// TIA Portal V20 export
FUNCTION "PlantAutoControl" : Void   // FC100, LAD
TITLE = Plant Automatic Control
// Per-equipment automatic-control layer for the shredding/material-recovery plant (REQ-001..022). Paradigm: combinational chained-permissive interlock/mapping (C-113 'no' - no phase memory in this block; the plant sequencer and equipment FBs hold the state). One network per machine, in material-train order, each mapping field feedback in, computing the auto start/shutdown permissives from PlantControl.Status and neighbour UPSEnable/ShutdownComplete, driving the physical output, and calling the equipment FB. Composed from the chained-permissive-enable pattern. Net 17 (feed conveyor) is freeform fwd/rev per C-116/C-117 (reversal pause enforced inside MotorFwdRevSystem). Author: lad-coder (gen-block-new). Rev 1, 2026-07-20.
BEGIN

REGION Network 1: Incline Feed Conveyor Automatic Control
   // Incline feed VSD (MotorVSDInst2). Running-fwd confirmation taken from the rotation sensor (inferred VSD-running mapping - review). Holds during shutdown until the link conveyor and the third-party JOB9001 plant have both completed shutdown (REQ-003/014); starts once the air-separator VSD is enabled (REQ-004).
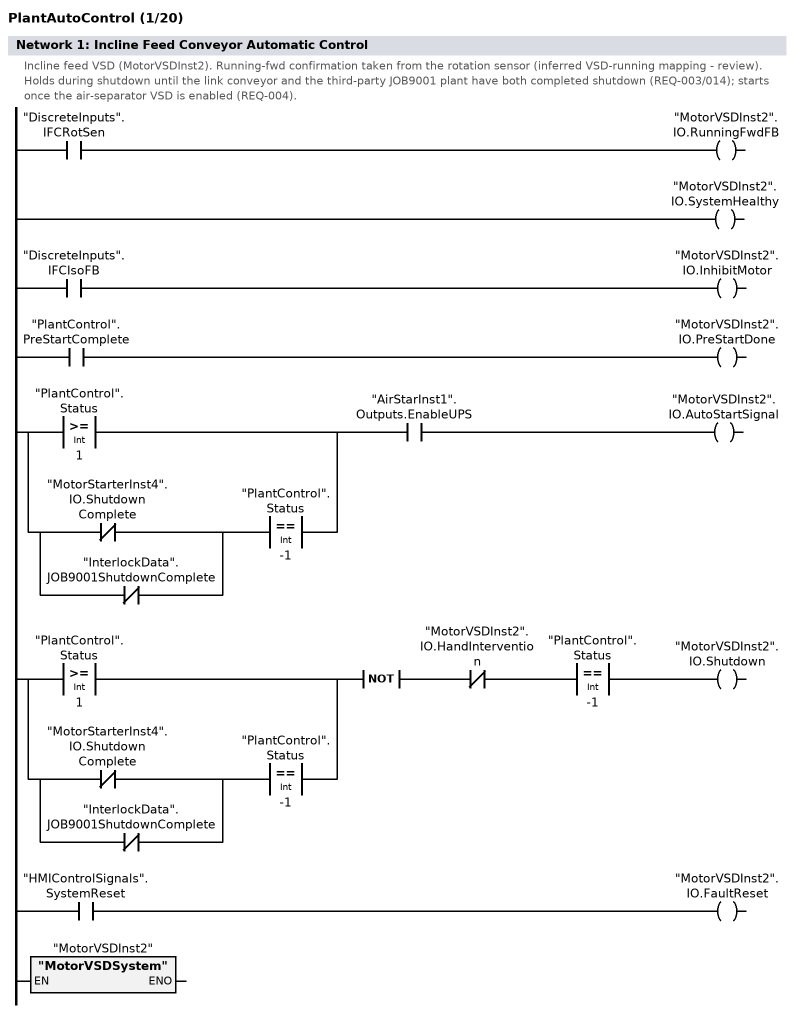
   "MotorVSDInst2".IO.RunningFwdFB := "DiscreteInputs".IFCRotSen;
   "MotorVSDInst2".IO.SystemHealthy := TRUE;
   "MotorVSDInst2".IO.InhibitMotor := "DiscreteInputs".IFCIsoFB;
   "MotorVSDInst2".IO.PreStartDone := "PlantControl".PreStartComplete;
   "MotorVSDInst2".IO.AutoStartSignal := (("PlantControl".Status >= 1) OR ((NOT "MotorStarterInst4".IO.ShutdownComplete OR NOT "InterlockData".JOB9001ShutdownComplete) AND ("PlantControl".Status = (-1)))) AND "AirStarInst1".Outputs.EnableUPS;
   "MotorVSDInst2".IO.Shutdown := NOT (("PlantControl".Status >= 1) OR ((NOT "MotorStarterInst4".IO.ShutdownComplete OR NOT "InterlockData".JOB9001ShutdownComplete) AND ("PlantControl".Status = (-1)))) AND NOT "MotorVSDInst2".IO.HandIntervention AND ("PlantControl".Status = (-1));
   "MotorVSDInst2".IO.FaultReset := "HMIControlSignals".SystemReset;
   "MotorVSDInst2"();   // "MotorVSDSystem"
END_REGION

REGION Network 2: Link Conveyor Automatic Control
   // Link conveyor (MotorStarterInst4), the designated first machine. Gated by the third-party JOB9001 interlock; holds through shutdown until JOB9001 signals its own shutdown complete (REQ-014). On first auto-start it requests the plant pre-start warning once (one-shot via PlantControl.PositiveEdgeArray[4]), cleared when the pre-start output energises (REQ-015).
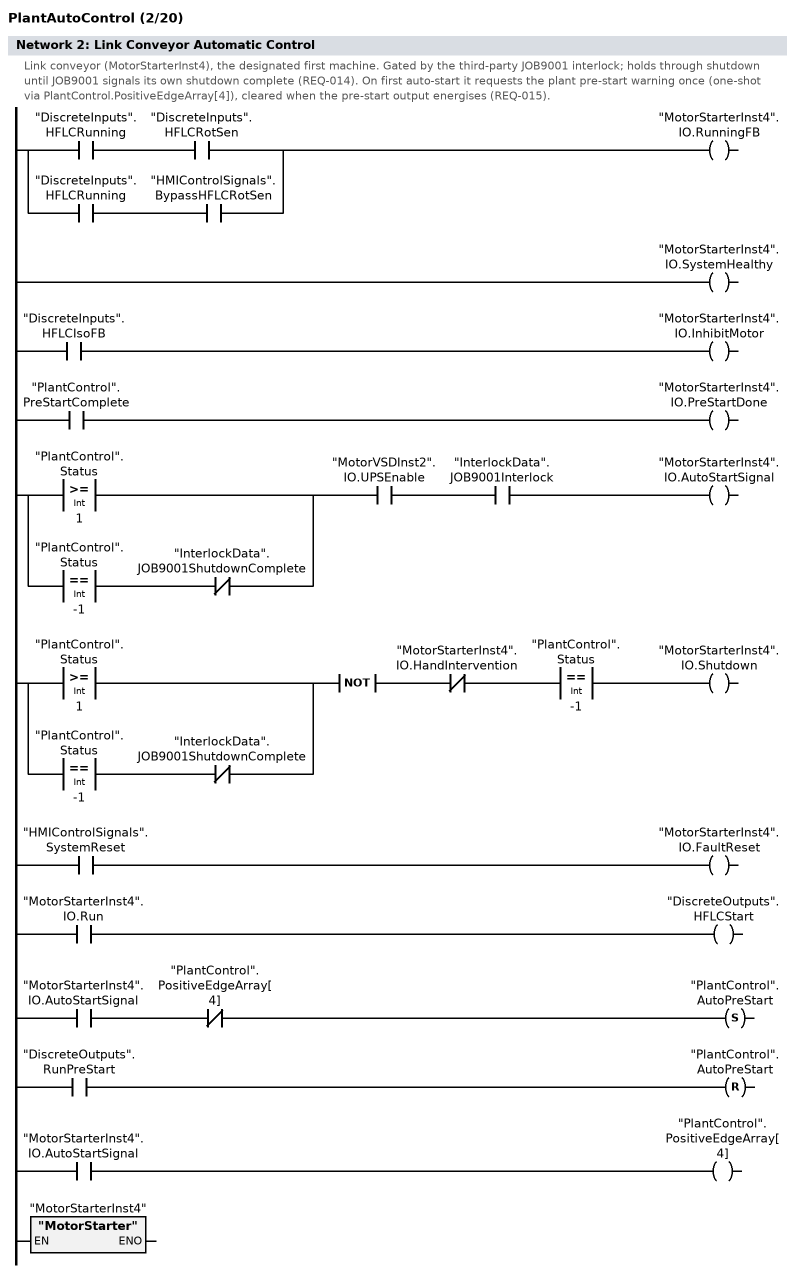
   "MotorStarterInst4".IO.RunningFB := ("DiscreteInputs".HFLCRunning AND "DiscreteInputs".HFLCRotSen) OR ("DiscreteInputs".HFLCRunning AND "HMIControlSignals".BypassHFLCRotSen);
   "MotorStarterInst4".IO.SystemHealthy := TRUE;
   "MotorStarterInst4".IO.InhibitMotor := "DiscreteInputs".HFLCIsoFB;
   "MotorStarterInst4".IO.PreStartDone := "PlantControl".PreStartComplete;
   "MotorStarterInst4".IO.AutoStartSignal := (("PlantControl".Status >= 1) OR (("PlantControl".Status = (-1)) AND NOT "InterlockData".JOB9001ShutdownComplete)) AND "MotorVSDInst2".IO.UPSEnable AND "InterlockData".JOB9001Interlock;
   "MotorStarterInst4".IO.Shutdown := NOT (("PlantControl".Status >= 1) OR (("PlantControl".Status = (-1)) AND NOT "InterlockData".JOB9001ShutdownComplete)) AND NOT "MotorStarterInst4".IO.HandIntervention AND ("PlantControl".Status = (-1));
   "MotorStarterInst4".IO.FaultReset := "HMIControlSignals".SystemReset;
   "DiscreteOutputs".HFLCStart := "MotorStarterInst4".IO.Run;
   IF "MotorStarterInst4".IO.AutoStartSignal AND NOT "PlantControl".PositiveEdgeArray[4] THEN
       "PlantControl".AutoPreStart := TRUE;
   END_IF;
   IF "DiscreteOutputs".RunPreStart THEN "PlantControl".AutoPreStart := FALSE; END_IF;
   "PlantControl".PositiveEdgeArray[4] := "MotorStarterInst4".IO.AutoStartSignal;
   "MotorStarterInst4"();   // "MotorStarter"
END_REGION

REGION Network 3: Dust Filter Unit 1 Automatic Control
   // Dust filter unit 1 (FilterUnitInst2). Remote-operational, running(=ready) and fault feedbacks brought in; fault reset echoed to the physical unit (REQ-019). Fan up-to-speed delay set from the plant fan-start time (REQ-020); see block header re C-308. Starts once the sorter conveyor VSD is enabled; holds during shutdown until fans-shutdown-ready (REQ-003/013).
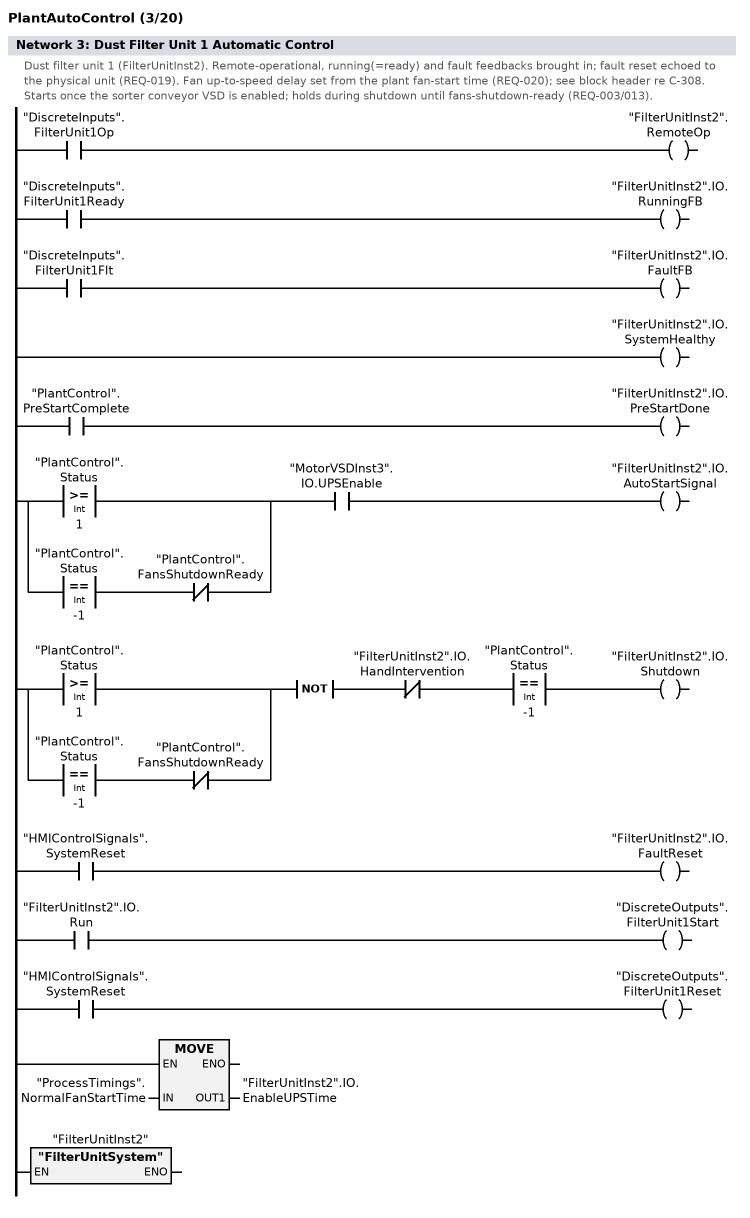
   "FilterUnitInst2".RemoteOp := "DiscreteInputs".FilterUnit1Op;
   "FilterUnitInst2".IO.RunningFB := "DiscreteInputs".FilterUnit1Ready;
   "FilterUnitInst2".IO.FaultFB := "DiscreteInputs".FilterUnit1Flt;
   "FilterUnitInst2".IO.SystemHealthy := TRUE;
   "FilterUnitInst2".IO.PreStartDone := "PlantControl".PreStartComplete;
   "FilterUnitInst2".IO.AutoStartSignal := (("PlantControl".Status >= 1) OR (("PlantControl".Status = (-1)) AND NOT "PlantControl".FansShutdownReady)) AND "MotorVSDInst3".IO.UPSEnable;
   "FilterUnitInst2".IO.Shutdown := NOT (("PlantControl".Status >= 1) OR (("PlantControl".Status = (-1)) AND NOT "PlantControl".FansShutdownReady)) AND NOT "FilterUnitInst2".IO.HandIntervention AND ("PlantControl".Status = (-1));
   "FilterUnitInst2".IO.FaultReset := "HMIControlSignals".SystemReset;
   "DiscreteOutputs".FilterUnit1Start := "FilterUnitInst2".IO.Run;
   "DiscreteOutputs".FilterUnit1Reset := "HMIControlSignals".SystemReset;
   "FilterUnitInst2".IO.EnableUPSTime := "ProcessTimings".NormalFanStartTime;
   "FilterUnitInst2"();   // "FilterUnitSystem"
END_REGION

REGION Network 4: Dust Filter Unit 2 Automatic Control
   // Dust filter unit 2 (FilterUnitInst3), identical shape to unit 1 (REQ-019/020). Starts once the sorter conveyor VSD is enabled; holds until fans-shutdown-ready.
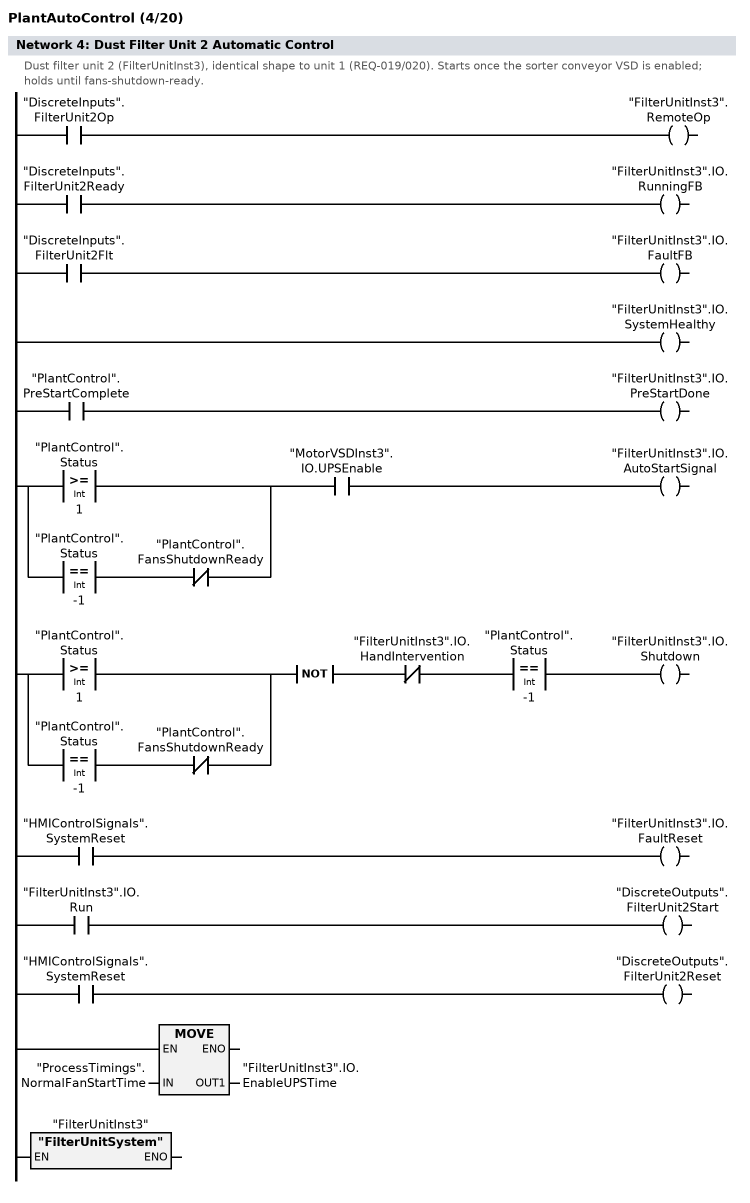
   "FilterUnitInst3".RemoteOp := "DiscreteInputs".FilterUnit2Op;
   "FilterUnitInst3".IO.RunningFB := "DiscreteInputs".FilterUnit2Ready;
   "FilterUnitInst3".IO.FaultFB := "DiscreteInputs".FilterUnit2Flt;
   "FilterUnitInst3".IO.SystemHealthy := TRUE;
   "FilterUnitInst3".IO.PreStartDone := "PlantControl".PreStartComplete;
   "FilterUnitInst3".IO.AutoStartSignal := (("PlantControl".Status >= 1) OR (("PlantControl".Status = (-1)) AND NOT "PlantControl".FansShutdownReady)) AND "MotorVSDInst3".IO.UPSEnable;
   "FilterUnitInst3".IO.Shutdown := NOT (("PlantControl".Status >= 1) OR (("PlantControl".Status = (-1)) AND NOT "PlantControl".FansShutdownReady)) AND NOT "FilterUnitInst3".IO.HandIntervention AND ("PlantControl".Status = (-1));
   "FilterUnitInst3".IO.FaultReset := "HMIControlSignals".SystemReset;
   "DiscreteOutputs".FilterUnit2Start := "FilterUnitInst3".IO.Run;
   "DiscreteOutputs".FilterUnit2Reset := "HMIControlSignals".SystemReset;
   "FilterUnitInst3".IO.EnableUPSTime := "ProcessTimings".NormalFanStartTime;
   "FilterUnitInst3"();   // "FilterUnitSystem"
END_REGION

REGION Network 5: Air-Separator VSD Automatic Control
   // Air-separator VSD (AirStarInst1), a bus-coupled drive with no discrete start output. Running confirmed over comms (MachineRunning). Alternative start permissive: discharge-conveyor VSD plus both dust filters enabled, OR discharge-conveyor VSD plus the third-party link-out signal (REQ-021). Holds during shutdown until the incline feed conveyor has shut down (REQ-003).
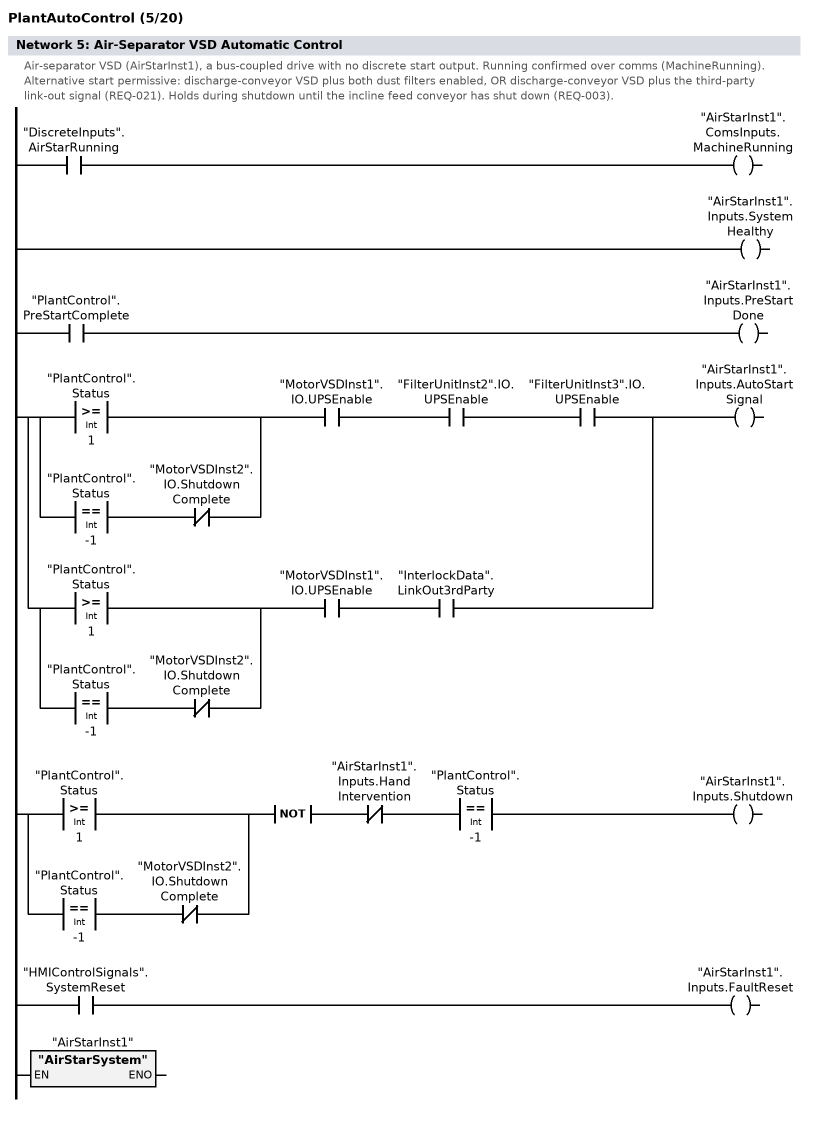
   "AirStarInst1".ComsInputs.MachineRunning := "DiscreteInputs".AirStarRunning;
   "AirStarInst1".Inputs.SystemHealthy := TRUE;
   "AirStarInst1".Inputs.PreStartDone := "PlantControl".PreStartComplete;
   "AirStarInst1".Inputs.AutoStartSignal := ((("PlantControl".Status >= 1) OR (("PlantControl".Status = (-1)) AND NOT "MotorVSDInst2".IO.ShutdownComplete)) AND "MotorVSDInst1".IO.UPSEnable AND "FilterUnitInst2".IO.UPSEnable AND "FilterUnitInst3".IO.UPSEnable) OR ((("PlantControl".Status >= 1) OR (("PlantControl".Status = (-1)) AND NOT "MotorVSDInst2".IO.ShutdownComplete)) AND "MotorVSDInst1".IO.UPSEnable AND "InterlockData".LinkOut3rdParty);
   "AirStarInst1".Inputs.Shutdown := NOT (("PlantControl".Status >= 1) OR (("PlantControl".Status = (-1)) AND NOT "MotorVSDInst2".IO.ShutdownComplete)) AND NOT "AirStarInst1".Inputs.HandIntervention AND ("PlantControl".Status = (-1));
   "AirStarInst1".Inputs.FaultReset := "HMIControlSignals".SystemReset;
   "AirStarInst1"();   // "AirStarSystem"
END_REGION

REGION Network 6: Discharge Conveyor VSD Automatic Control
   // Discharge conveyor VSD (MotorVSDInst1). Treats its rotation sensor as running-forward confirmation (REQ-012; bypass handling deferred - review). Starts once the overband magnet and ECS are enabled; holds during shutdown until the air-separator VSD has shut down (REQ-003/004).
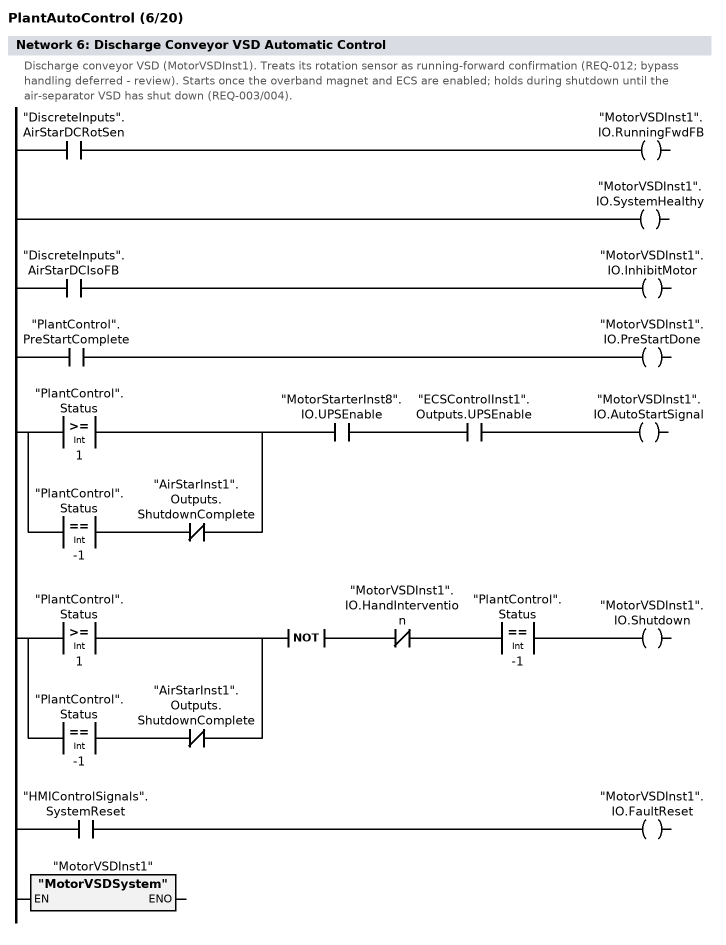
   "MotorVSDInst1".IO.RunningFwdFB := "DiscreteInputs".AirStarDCRotSen;
   "MotorVSDInst1".IO.SystemHealthy := TRUE;
   "MotorVSDInst1".IO.InhibitMotor := "DiscreteInputs".AirStarDCIsoFB;
   "MotorVSDInst1".IO.PreStartDone := "PlantControl".PreStartComplete;
   "MotorVSDInst1".IO.AutoStartSignal := (("PlantControl".Status >= 1) OR (("PlantControl".Status = (-1)) AND NOT "AirStarInst1".Outputs.ShutdownComplete)) AND "MotorStarterInst8".IO.UPSEnable AND "ECSControlInst1".Outputs.UPSEnable;
   "MotorVSDInst1".IO.Shutdown := NOT (("PlantControl".Status >= 1) OR (("PlantControl".Status = (-1)) AND NOT "AirStarInst1".Outputs.ShutdownComplete)) AND NOT "MotorVSDInst1".IO.HandIntervention AND ("PlantControl".Status = (-1));
   "MotorVSDInst1".IO.FaultReset := "HMIControlSignals".SystemReset;
   "MotorVSDInst1"();   // "MotorVSDSystem"
END_REGION

REGION Network 7: Metal Collection Conveyor Automatic Control
   // Metal collection conveyor (MotorStarterInst3). Gated by the magnet-circuit enable (REQ-013); starts on that plant flag rather than an upstream UPSEnable. Holds during shutdown until the overband magnet has shut down (REQ-003).
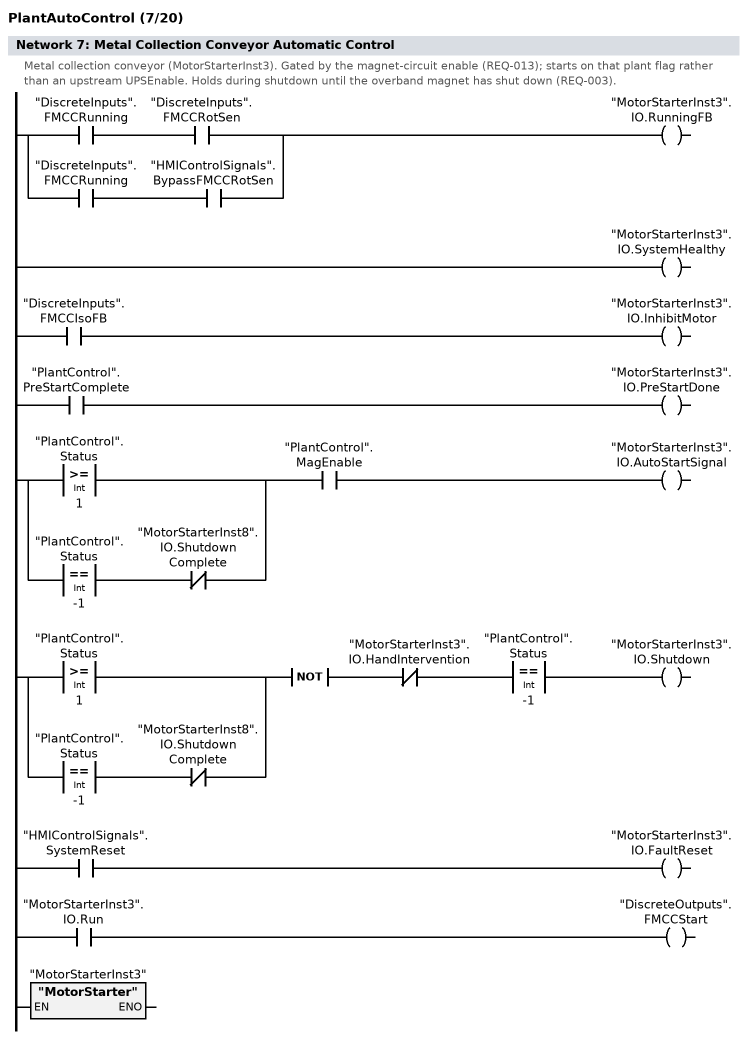
   "MotorStarterInst3".IO.RunningFB := ("DiscreteInputs".FMCCRunning AND "DiscreteInputs".FMCCRotSen) OR ("DiscreteInputs".FMCCRunning AND "HMIControlSignals".BypassFMCCRotSen);
   "MotorStarterInst3".IO.SystemHealthy := TRUE;
   "MotorStarterInst3".IO.InhibitMotor := "DiscreteInputs".FMCCIsoFB;
   "MotorStarterInst3".IO.PreStartDone := "PlantControl".PreStartComplete;
   "MotorStarterInst3".IO.AutoStartSignal := (("PlantControl".Status >= 1) OR (("PlantControl".Status = (-1)) AND NOT "MotorStarterInst8".IO.ShutdownComplete)) AND "PlantControl".MagEnable;
   "MotorStarterInst3".IO.Shutdown := NOT (("PlantControl".Status >= 1) OR (("PlantControl".Status = (-1)) AND NOT "MotorStarterInst8".IO.ShutdownComplete)) AND NOT "MotorStarterInst3".IO.HandIntervention AND ("PlantControl".Status = (-1));
   "MotorStarterInst3".IO.FaultReset := "HMIControlSignals".SystemReset;
   "DiscreteOutputs".FMCCStart := "MotorStarterInst3".IO.Run;
   "MotorStarterInst3"();   // "MotorStarter"
END_REGION

REGION Network 8: Overband Magnet Automatic Control
   // Overband magnet (MotorStarterInst8), confirmed on run feedback only (no rotation sensor). Starts once the metal collection conveyor is enabled; holds during shutdown until the discharge conveyor VSD has shut down (REQ-003/004).
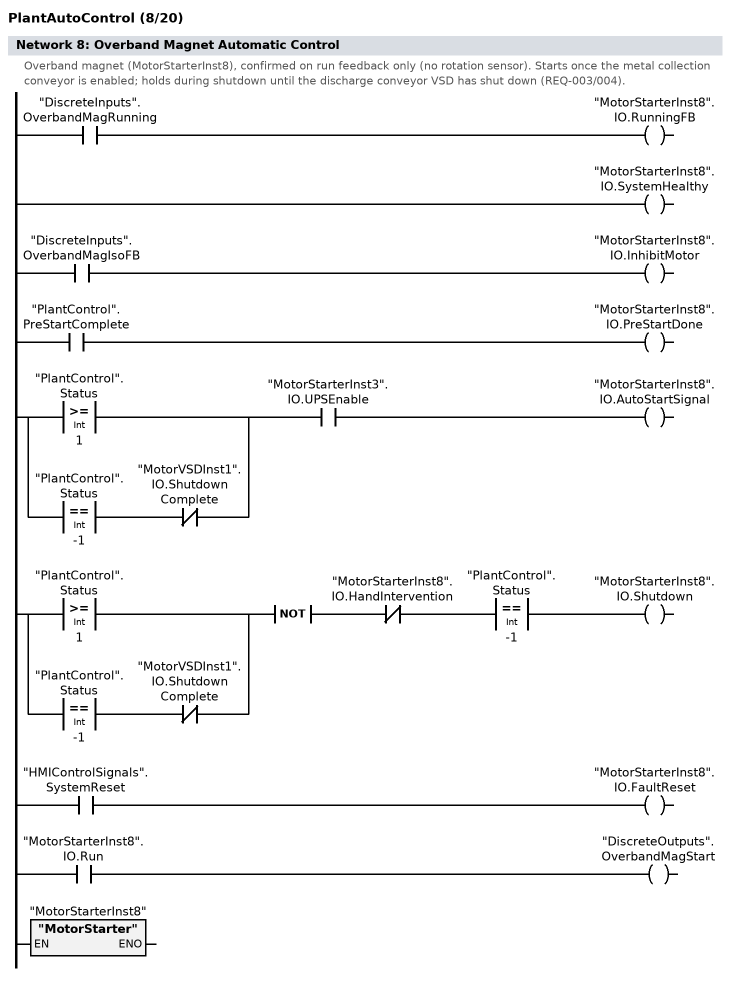
   "MotorStarterInst8".IO.RunningFB := "DiscreteInputs".OverbandMagRunning;
   "MotorStarterInst8".IO.SystemHealthy := TRUE;
   "MotorStarterInst8".IO.InhibitMotor := "DiscreteInputs".OverbandMagIsoFB;
   "MotorStarterInst8".IO.PreStartDone := "PlantControl".PreStartComplete;
   "MotorStarterInst8".IO.AutoStartSignal := (("PlantControl".Status >= 1) OR (("PlantControl".Status = (-1)) AND NOT "MotorVSDInst1".IO.ShutdownComplete)) AND "MotorStarterInst3".IO.UPSEnable;
   "MotorStarterInst8".IO.Shutdown := NOT (("PlantControl".Status >= 1) OR (("PlantControl".Status = (-1)) AND NOT "MotorVSDInst1".IO.ShutdownComplete)) AND NOT "MotorStarterInst8".IO.HandIntervention AND ("PlantControl".Status = (-1));
   "MotorStarterInst8".IO.FaultReset := "HMIControlSignals".SystemReset;
   "DiscreteOutputs".OverbandMagStart := "MotorStarterInst8".IO.Run;
   "MotorStarterInst8"();   // "MotorStarter"
END_REGION

REGION Network 9: Equipment Control System Automatic Control
   // Equipment control system (ECSControlInst1). Fault, mode (auto/hand/setting), ready, running, feeder/charge and rotor status brought in; auto-start and reset outputs driven (REQ-018). Starts once the sorter conveyor VSD is enabled; holds during shutdown until the discharge conveyor VSD has shut down (REQ-003).
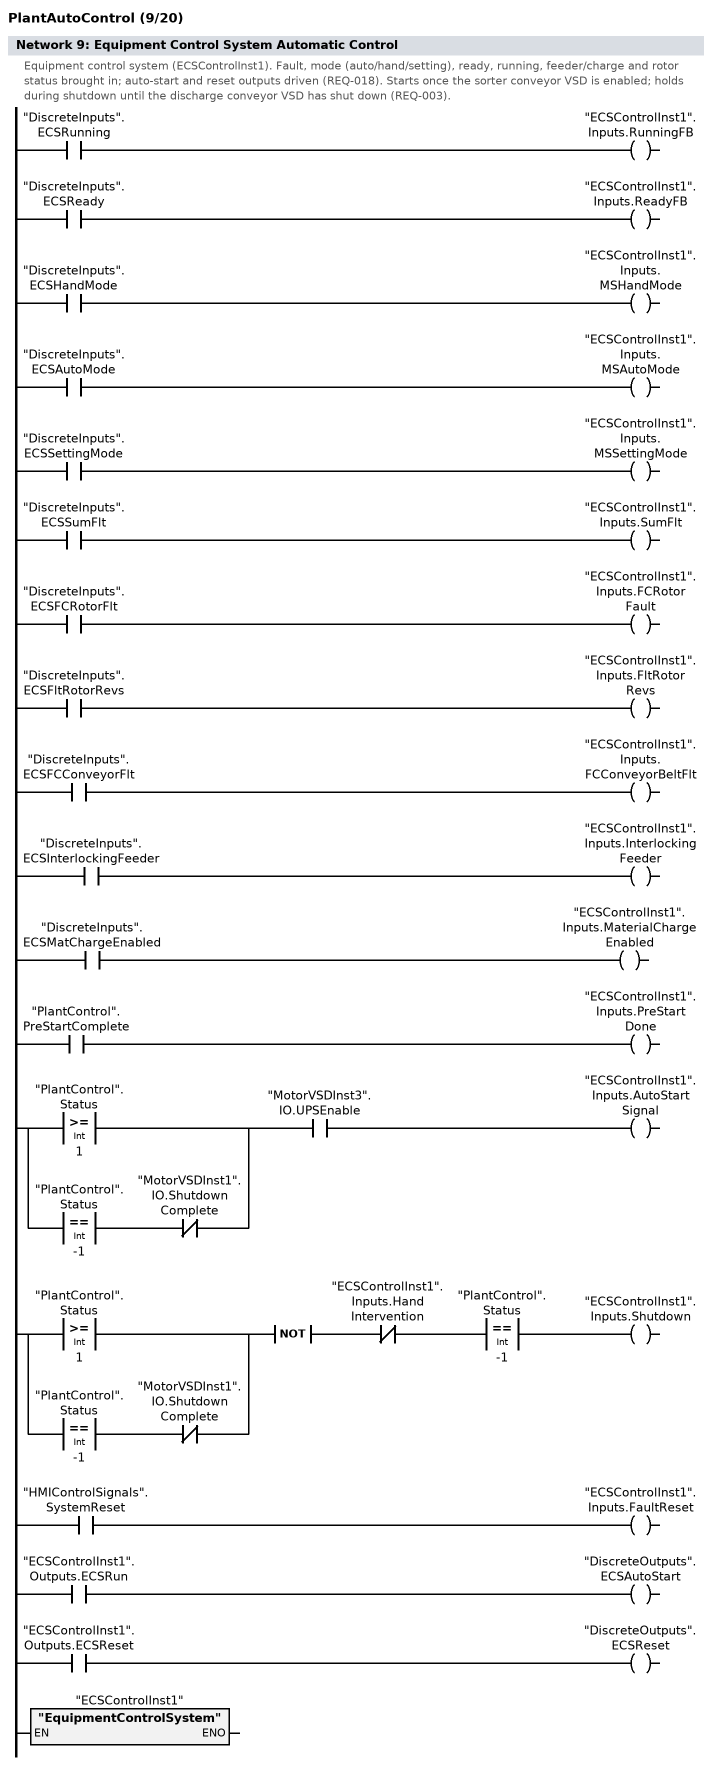
   "ECSControlInst1".Inputs.RunningFB := "DiscreteInputs".ECSRunning;
   "ECSControlInst1".Inputs.ReadyFB := "DiscreteInputs".ECSReady;
   "ECSControlInst1".Inputs.MSHandMode := "DiscreteInputs".ECSHandMode;
   "ECSControlInst1".Inputs.MSAutoMode := "DiscreteInputs".ECSAutoMode;
   "ECSControlInst1".Inputs.MSSettingMode := "DiscreteInputs".ECSSettingMode;
   "ECSControlInst1".Inputs.SumFlt := "DiscreteInputs".ECSSumFlt;
   "ECSControlInst1".Inputs.FCRotorFault := "DiscreteInputs".ECSFCRotorFlt;
   "ECSControlInst1".Inputs.FltRotorRevs := "DiscreteInputs".ECSFltRotorRevs;
   "ECSControlInst1".Inputs.FCConveyorBeltFlt := "DiscreteInputs".ECSFCConveyorFlt;
   "ECSControlInst1".Inputs.InterlockingFeeder := "DiscreteInputs".ECSInterlockingFeeder;
   "ECSControlInst1".Inputs.MaterialChargeEnabled := "DiscreteInputs".ECSMatChargeEnabled;
   "ECSControlInst1".Inputs.PreStartDone := "PlantControl".PreStartComplete;
   "ECSControlInst1".Inputs.AutoStartSignal := (("PlantControl".Status >= 1) OR (("PlantControl".Status = (-1)) AND NOT "MotorVSDInst1".IO.ShutdownComplete)) AND "MotorVSDInst3".IO.UPSEnable;
   "ECSControlInst1".Inputs.Shutdown := NOT (("PlantControl".Status >= 1) OR (("PlantControl".Status = (-1)) AND NOT "MotorVSDInst1".IO.ShutdownComplete)) AND NOT "ECSControlInst1".Inputs.HandIntervention AND ("PlantControl".Status = (-1));
   "ECSControlInst1".Inputs.FaultReset := "HMIControlSignals".SystemReset;
   "DiscreteOutputs".ECSAutoStart := "ECSControlInst1".Outputs.ECSRun;
   "DiscreteOutputs".ECSReset := "ECSControlInst1".Outputs.ECSReset;
   "ECSControlInst1"();   // "EquipmentControlSystem"
END_REGION

REGION Network 10: Sorter Conveyor VSD Automatic Control
   // Sorter feed conveyor VSD (MotorVSDInst3). Running-fwd from rotation sensor (inferred - review). Only permitted to start while the optical sorter is ready and not faulted, and the ejected and residual conveyors are enabled (REQ-017/004). Holds during shutdown until the ECS has shut down (REQ-003).
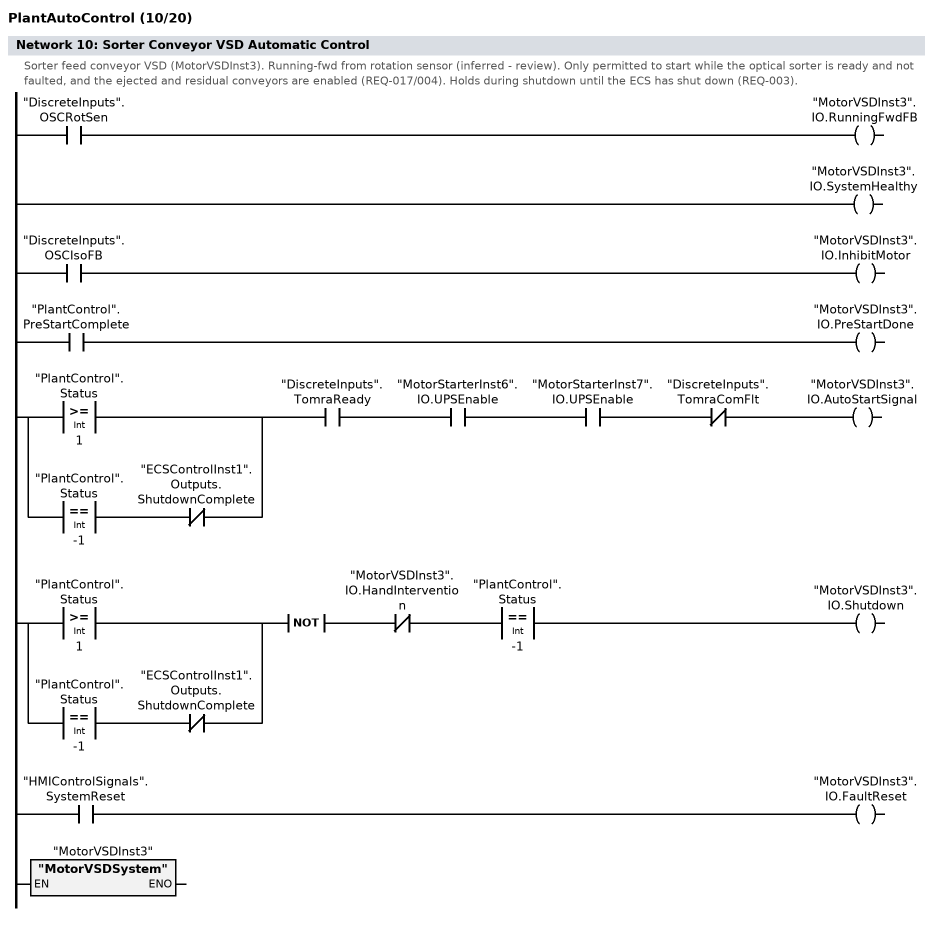
   "MotorVSDInst3".IO.RunningFwdFB := "DiscreteInputs".OSCRotSen;
   "MotorVSDInst3".IO.SystemHealthy := TRUE;
   "MotorVSDInst3".IO.InhibitMotor := "DiscreteInputs".OSCIsoFB;
   "MotorVSDInst3".IO.PreStartDone := "PlantControl".PreStartComplete;
   "MotorVSDInst3".IO.AutoStartSignal := (("PlantControl".Status >= 1) OR (("PlantControl".Status = (-1)) AND NOT "ECSControlInst1".Outputs.ShutdownComplete)) AND "DiscreteInputs".TomraReady AND "MotorStarterInst6".IO.UPSEnable AND "MotorStarterInst7".IO.UPSEnable AND NOT "DiscreteInputs".TomraComFlt;
   "MotorVSDInst3".IO.Shutdown := NOT (("PlantControl".Status >= 1) OR (("PlantControl".Status = (-1)) AND NOT "ECSControlInst1".Outputs.ShutdownComplete)) AND NOT "MotorVSDInst3".IO.HandIntervention AND ("PlantControl".Status = (-1));
   "MotorVSDInst3".IO.FaultReset := "HMIControlSignals".SystemReset;
   "MotorVSDInst3"();   // "MotorVSDSystem"
END_REGION

REGION Network 11: Optical Sorter Automatic Control
   // Optical sorter (TomraControlInst1). Hardwired ready/running/comms-fault brought in and the run command driven to the sorter (REQ-017). Comms data words (a separate block owns them) deliberately not wired here. Starts once the ejected and residual conveyors are enabled; holds during shutdown until the sorter conveyor VSD has shut down (REQ-003).
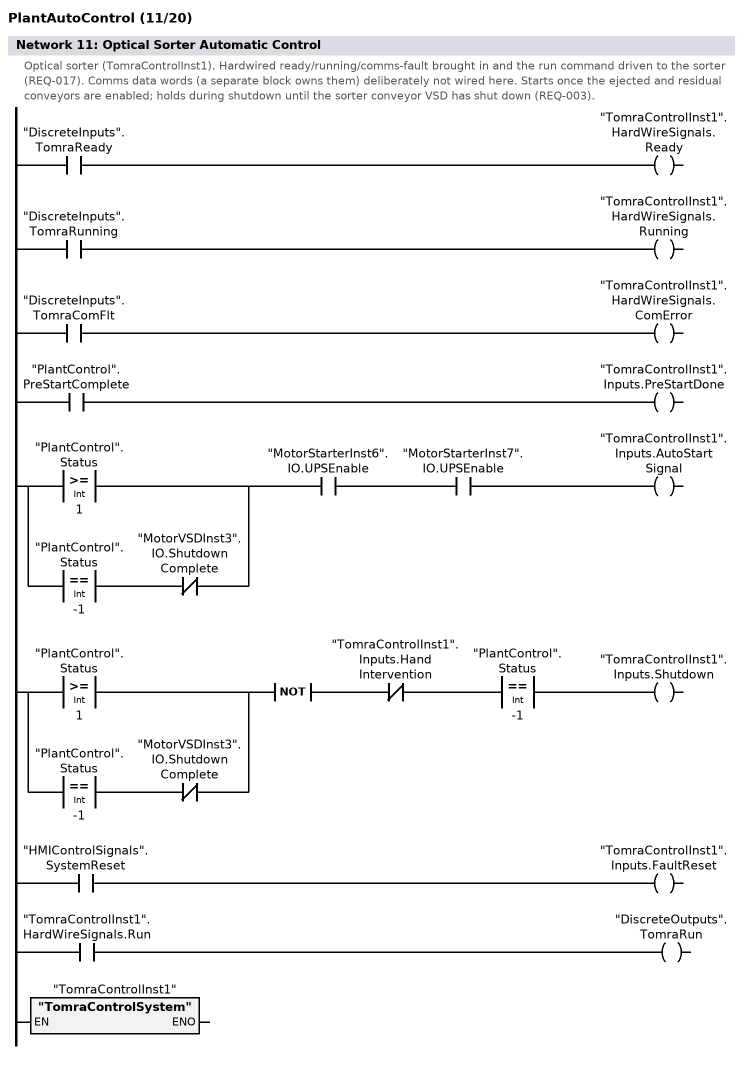
   "TomraControlInst1".HardWireSignals.Ready := "DiscreteInputs".TomraReady;
   "TomraControlInst1".HardWireSignals.Running := "DiscreteInputs".TomraRunning;
   "TomraControlInst1".HardWireSignals.ComError := "DiscreteInputs".TomraComFlt;
   "TomraControlInst1".Inputs.PreStartDone := "PlantControl".PreStartComplete;
   "TomraControlInst1".Inputs.AutoStartSignal := (("PlantControl".Status >= 1) OR (("PlantControl".Status = (-1)) AND NOT "MotorVSDInst3".IO.ShutdownComplete)) AND "MotorStarterInst6".IO.UPSEnable AND "MotorStarterInst7".IO.UPSEnable;
   "TomraControlInst1".Inputs.Shutdown := NOT (("PlantControl".Status >= 1) OR (("PlantControl".Status = (-1)) AND NOT "MotorVSDInst3".IO.ShutdownComplete)) AND NOT "TomraControlInst1".Inputs.HandIntervention AND ("PlantControl".Status = (-1));
   "TomraControlInst1".Inputs.FaultReset := "HMIControlSignals".SystemReset;
   "DiscreteOutputs".TomraRun := "TomraControlInst1".HardWireSignals.Run;
   "TomraControlInst1"();   // "TomraControlSystem"
END_REGION

REGION Network 12: Drum Separator Automatic Control
   // Drum separator (MotorStarterInst5), confirmed on run feedback only. Gated by the drum-separator enable (REQ-013); holds during shutdown until drum-shutdown-ready (REQ-003).
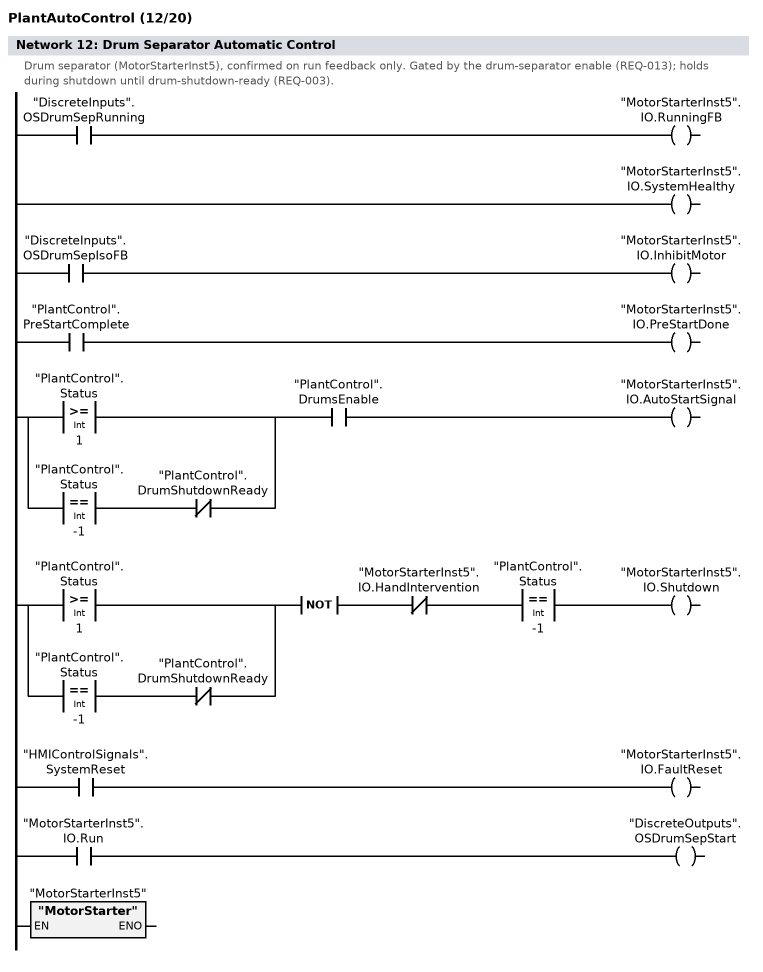
   "MotorStarterInst5".IO.RunningFB := "DiscreteInputs".OSDrumSepRunning;
   "MotorStarterInst5".IO.SystemHealthy := TRUE;
   "MotorStarterInst5".IO.InhibitMotor := "DiscreteInputs".OSDrumSepIsoFB;
   "MotorStarterInst5".IO.PreStartDone := "PlantControl".PreStartComplete;
   "MotorStarterInst5".IO.AutoStartSignal := (("PlantControl".Status >= 1) OR (("PlantControl".Status = (-1)) AND NOT "PlantControl".DrumShutdownReady)) AND "PlantControl".DrumsEnable;
   "MotorStarterInst5".IO.Shutdown := NOT (("PlantControl".Status >= 1) OR (("PlantControl".Status = (-1)) AND NOT "PlantControl".DrumShutdownReady)) AND NOT "MotorStarterInst5".IO.HandIntervention AND ("PlantControl".Status = (-1));
   "MotorStarterInst5".IO.FaultReset := "HMIControlSignals".SystemReset;
   "DiscreteOutputs".OSDrumSepStart := "MotorStarterInst5".IO.Run;
   "MotorStarterInst5"();   // "MotorStarter"
END_REGION

REGION Network 13: Ejected Material Conveyor Automatic Control
   // Ejected material conveyor (MotorStarterInst6). Gated by the general enable (REQ-013); holds during shutdown until the optical sorter has shut down (REQ-003).
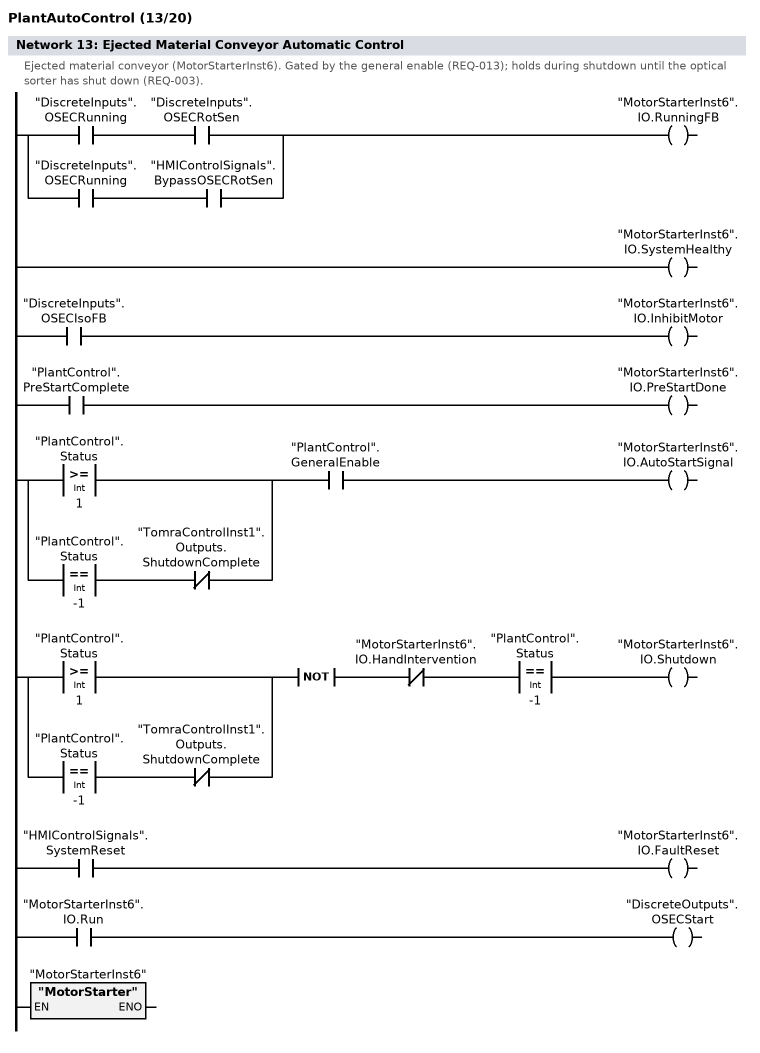
   "MotorStarterInst6".IO.RunningFB := ("DiscreteInputs".OSECRunning AND "DiscreteInputs".OSECRotSen) OR ("DiscreteInputs".OSECRunning AND "HMIControlSignals".BypassOSECRotSen);
   "MotorStarterInst6".IO.SystemHealthy := TRUE;
   "MotorStarterInst6".IO.InhibitMotor := "DiscreteInputs".OSECIsoFB;
   "MotorStarterInst6".IO.PreStartDone := "PlantControl".PreStartComplete;
   "MotorStarterInst6".IO.AutoStartSignal := (("PlantControl".Status >= 1) OR (("PlantControl".Status = (-1)) AND NOT "TomraControlInst1".Outputs.ShutdownComplete)) AND "PlantControl".GeneralEnable;
   "MotorStarterInst6".IO.Shutdown := NOT (("PlantControl".Status >= 1) OR (("PlantControl".Status = (-1)) AND NOT "TomraControlInst1".Outputs.ShutdownComplete)) AND NOT "MotorStarterInst6".IO.HandIntervention AND ("PlantControl".Status = (-1));
   "MotorStarterInst6".IO.FaultReset := "HMIControlSignals".SystemReset;
   "DiscreteOutputs".OSECStart := "MotorStarterInst6".IO.Run;
   "MotorStarterInst6"();   // "MotorStarter"
END_REGION

REGION Network 14: Residual Material Conveyor Automatic Control
   // Residual material conveyor (MotorStarterInst7). Starts once disc spreaders 1 and 2 are enabled; holds during shutdown until the optical sorter has shut down (REQ-003/004).
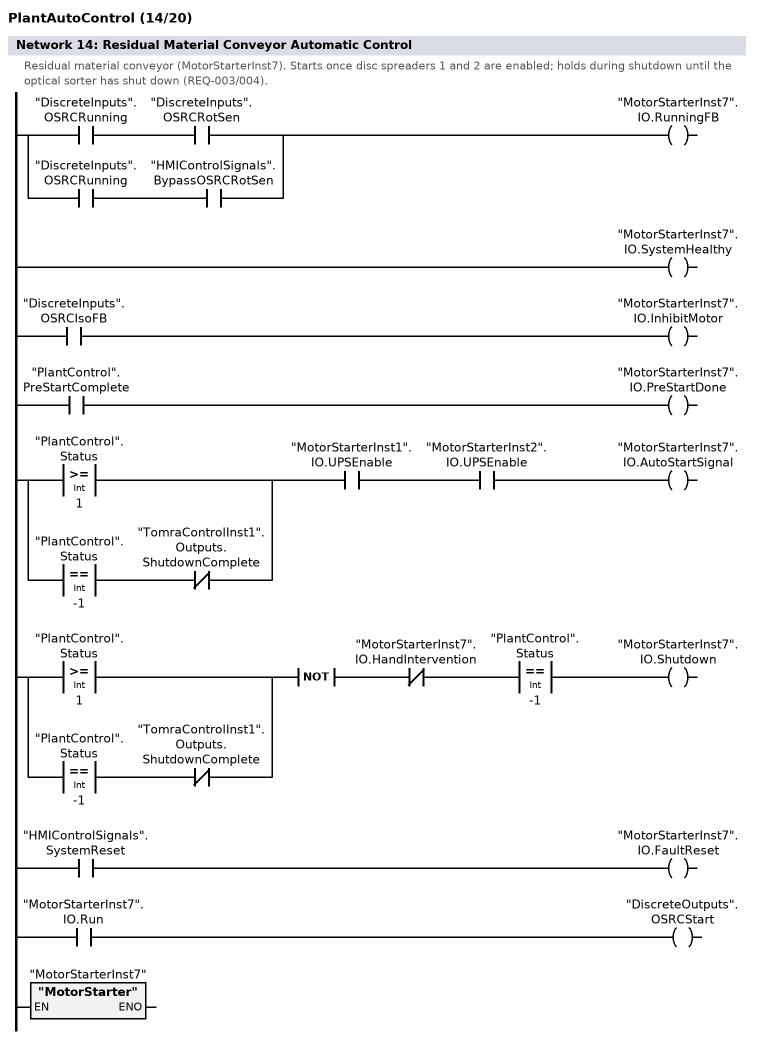
   "MotorStarterInst7".IO.RunningFB := ("DiscreteInputs".OSRCRunning AND "DiscreteInputs".OSRCRotSen) OR ("DiscreteInputs".OSRCRunning AND "HMIControlSignals".BypassOSRCRotSen);
   "MotorStarterInst7".IO.SystemHealthy := TRUE;
   "MotorStarterInst7".IO.InhibitMotor := "DiscreteInputs".OSRCIsoFB;
   "MotorStarterInst7".IO.PreStartDone := "PlantControl".PreStartComplete;
   "MotorStarterInst7".IO.AutoStartSignal := (("PlantControl".Status >= 1) OR (("PlantControl".Status = (-1)) AND NOT "TomraControlInst1".Outputs.ShutdownComplete)) AND "MotorStarterInst1".IO.UPSEnable AND "MotorStarterInst2".IO.UPSEnable;
   "MotorStarterInst7".IO.Shutdown := NOT (("PlantControl".Status >= 1) OR (("PlantControl".Status = (-1)) AND NOT "TomraControlInst1".Outputs.ShutdownComplete)) AND NOT "MotorStarterInst7".IO.HandIntervention AND ("PlantControl".Status = (-1));
   "MotorStarterInst7".IO.FaultReset := "HMIControlSignals".SystemReset;
   "DiscreteOutputs".OSRCStart := "MotorStarterInst7".IO.Run;
   "MotorStarterInst7"();   // "MotorStarter"
END_REGION

REGION Network 15: Disc Spreader Unit 1 Automatic Control
   // Disc spreader unit 1 (MotorStarterInst1), confirmed on run feedback only. Starts once the feed conveyor is enabled; holds during shutdown until the residual material conveyor has shut down (REQ-003/004).
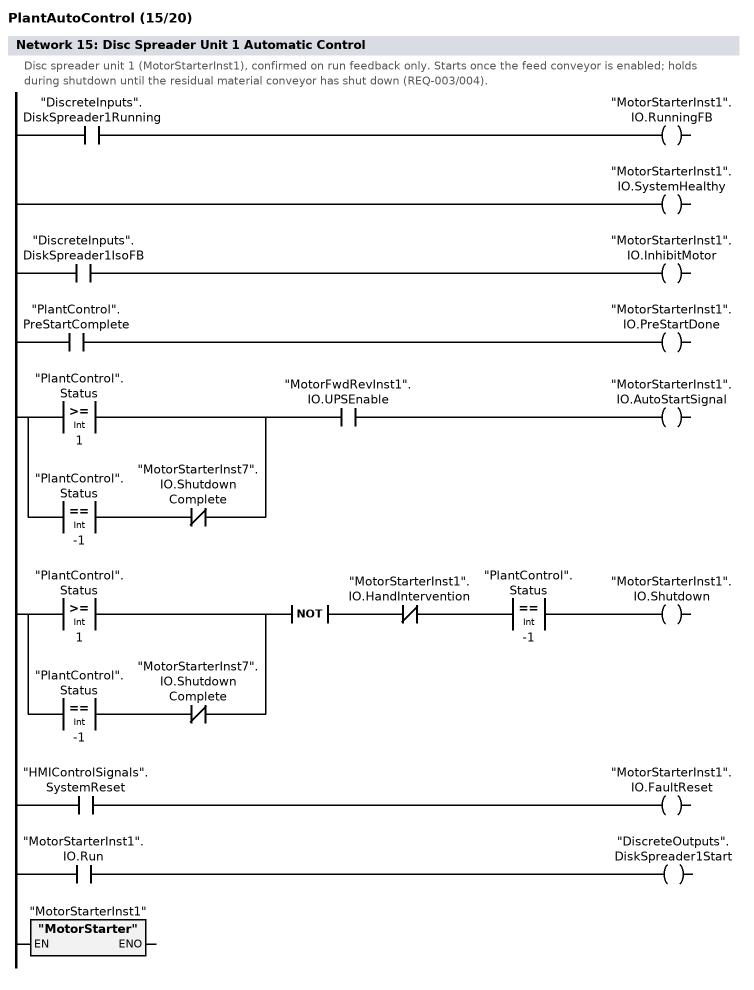
   "MotorStarterInst1".IO.RunningFB := "DiscreteInputs".DiskSpreader1Running;
   "MotorStarterInst1".IO.SystemHealthy := TRUE;
   "MotorStarterInst1".IO.InhibitMotor := "DiscreteInputs".DiskSpreader1IsoFB;
   "MotorStarterInst1".IO.PreStartDone := "PlantControl".PreStartComplete;
   "MotorStarterInst1".IO.AutoStartSignal := (("PlantControl".Status >= 1) OR (("PlantControl".Status = (-1)) AND NOT "MotorStarterInst7".IO.ShutdownComplete)) AND "MotorFwdRevInst1".IO.UPSEnable;
   "MotorStarterInst1".IO.Shutdown := NOT (("PlantControl".Status >= 1) OR (("PlantControl".Status = (-1)) AND NOT "MotorStarterInst7".IO.ShutdownComplete)) AND NOT "MotorStarterInst1".IO.HandIntervention AND ("PlantControl".Status = (-1));
   "MotorStarterInst1".IO.FaultReset := "HMIControlSignals".SystemReset;
   "DiscreteOutputs".DiskSpreader1Start := "MotorStarterInst1".IO.Run;
   "MotorStarterInst1"();   // "MotorStarter"
END_REGION

REGION Network 16: Disc Spreader Unit 2 Automatic Control
   // Disc spreader unit 2 (MotorStarterInst2), identical shape to unit 1. Starts once the feed conveyor is enabled; holds until the residual material conveyor has shut down (REQ-003/004).
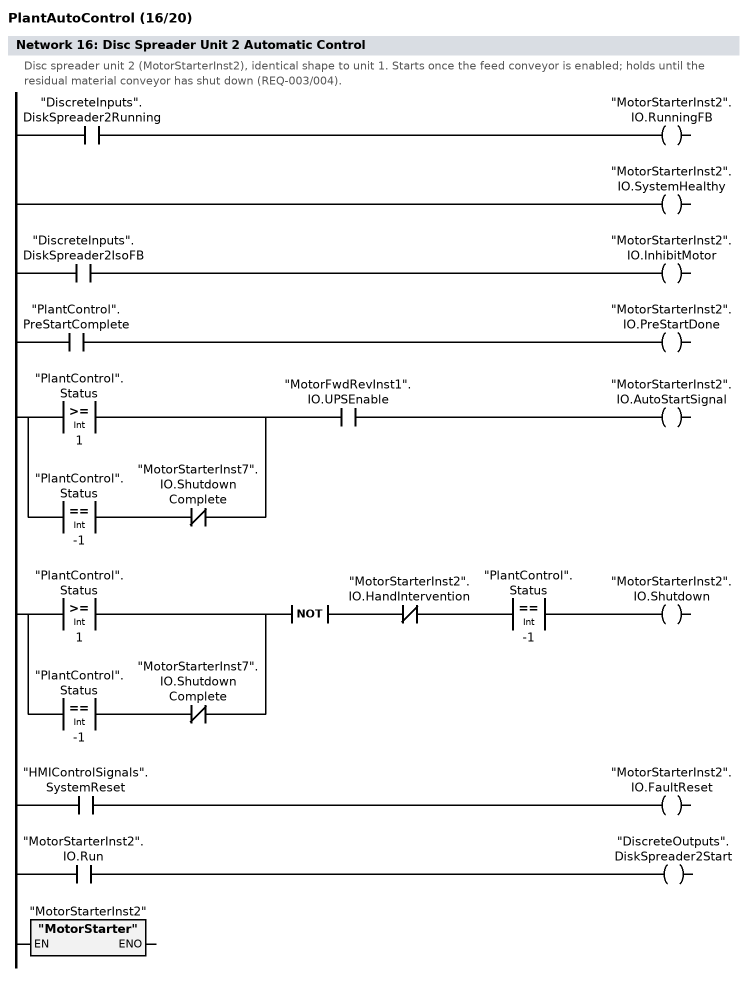
   "MotorStarterInst2".IO.RunningFB := "DiscreteInputs".DiskSpreader2Running;
   "MotorStarterInst2".IO.SystemHealthy := TRUE;
   "MotorStarterInst2".IO.InhibitMotor := "DiscreteInputs".DiskSpreader2IsoFB;
   "MotorStarterInst2".IO.PreStartDone := "PlantControl".PreStartComplete;
   "MotorStarterInst2".IO.AutoStartSignal := (("PlantControl".Status >= 1) OR (("PlantControl".Status = (-1)) AND NOT "MotorStarterInst7".IO.ShutdownComplete)) AND "MotorFwdRevInst1".IO.UPSEnable;
   "MotorStarterInst2".IO.Shutdown := NOT (("PlantControl".Status >= 1) OR (("PlantControl".Status = (-1)) AND NOT "MotorStarterInst7".IO.ShutdownComplete)) AND NOT "MotorStarterInst2".IO.HandIntervention AND ("PlantControl".Status = (-1));
   "MotorStarterInst2".IO.FaultReset := "HMIControlSignals".SystemReset;
   "DiscreteOutputs".DiskSpreader2Start := "MotorStarterInst2".IO.Run;
   "MotorStarterInst2"();   // "MotorStarter"
END_REGION

REGION Network 17: Feed Conveyor Automatic Control
   // Shredder feed conveyor (MotorFwdRevInst1), forward/reverse. Runs forward when the shredder is ready to receive (its upstream-enable), reverses on the general enable to back material off the shredder when it is not ready (REQ-016). Reverse selection is FREEFORM (no admitted pattern for fwd/rev); the stopped-before-reverse pause is enforced inside MotorFwdRevSystem (C-117). Holds during shutdown until disc spreaders 1 and 2 have shut down (REQ-003).
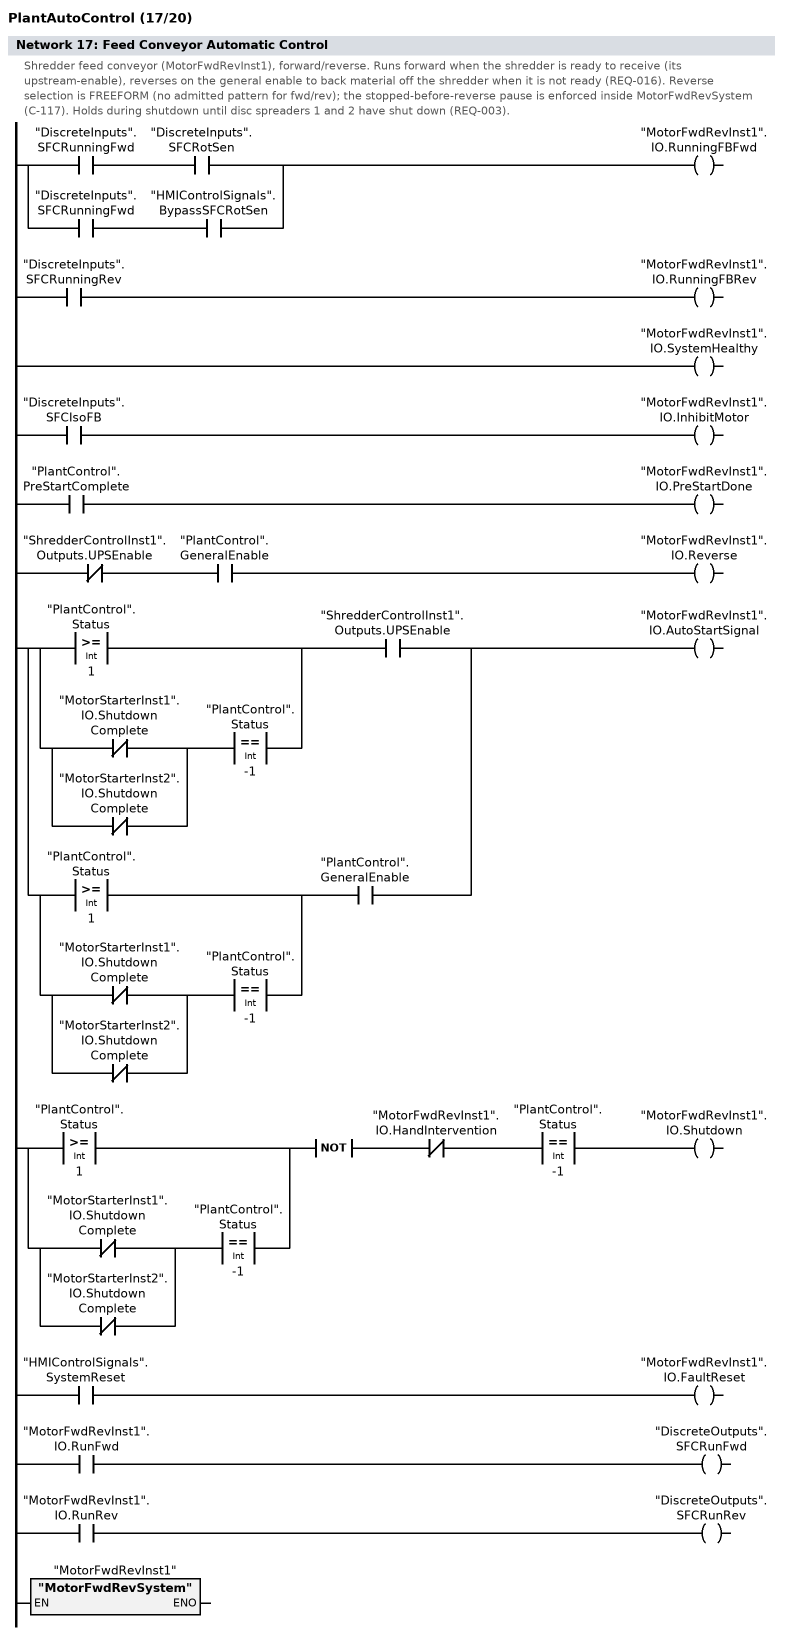
   "MotorFwdRevInst1".IO.RunningFBFwd := ("DiscreteInputs".SFCRunningFwd AND "DiscreteInputs".SFCRotSen) OR ("DiscreteInputs".SFCRunningFwd AND "HMIControlSignals".BypassSFCRotSen);
   "MotorFwdRevInst1".IO.RunningFBRev := "DiscreteInputs".SFCRunningRev;
   "MotorFwdRevInst1".IO.SystemHealthy := TRUE;
   "MotorFwdRevInst1".IO.InhibitMotor := "DiscreteInputs".SFCIsoFB;
   "MotorFwdRevInst1".IO.PreStartDone := "PlantControl".PreStartComplete;
   "MotorFwdRevInst1".IO.Reverse := NOT "ShredderControlInst1".Outputs.UPSEnable AND "PlantControl".GeneralEnable;
   "MotorFwdRevInst1".IO.AutoStartSignal := ((("PlantControl".Status >= 1) OR ((NOT "MotorStarterInst1".IO.ShutdownComplete OR NOT "MotorStarterInst2".IO.ShutdownComplete) AND ("PlantControl".Status = (-1)))) AND "ShredderControlInst1".Outputs.UPSEnable) OR ((("PlantControl".Status >= 1) OR ((NOT "MotorStarterInst1".IO.ShutdownComplete OR NOT "MotorStarterInst2".IO.ShutdownComplete) AND ("PlantControl".Status = (-1)))) AND "PlantControl".GeneralEnable);
   "MotorFwdRevInst1".IO.Shutdown := NOT (("PlantControl".Status >= 1) OR ((NOT "MotorStarterInst1".IO.ShutdownComplete OR NOT "MotorStarterInst2".IO.ShutdownComplete) AND ("PlantControl".Status = (-1)))) AND NOT "MotorFwdRevInst1".IO.HandIntervention AND ("PlantControl".Status = (-1));
   "MotorFwdRevInst1".IO.FaultReset := "HMIControlSignals".SystemReset;
   "DiscreteOutputs".SFCRunFwd := "MotorFwdRevInst1".IO.RunFwd;
   "DiscreteOutputs".SFCRunRev := "MotorFwdRevInst1".IO.RunRev;
   "MotorFwdRevInst1"();   // "MotorFwdRevSystem"
END_REGION

REGION Network 18: Shredder Automatic Control
   // Shredder (ShredderControlInst1), commanded through its FB (no discrete start; internal sequence out of scope). Starts once the discharge conveyor is enabled; holds during shutdown until the feed conveyor has shut down (REQ-003/004).
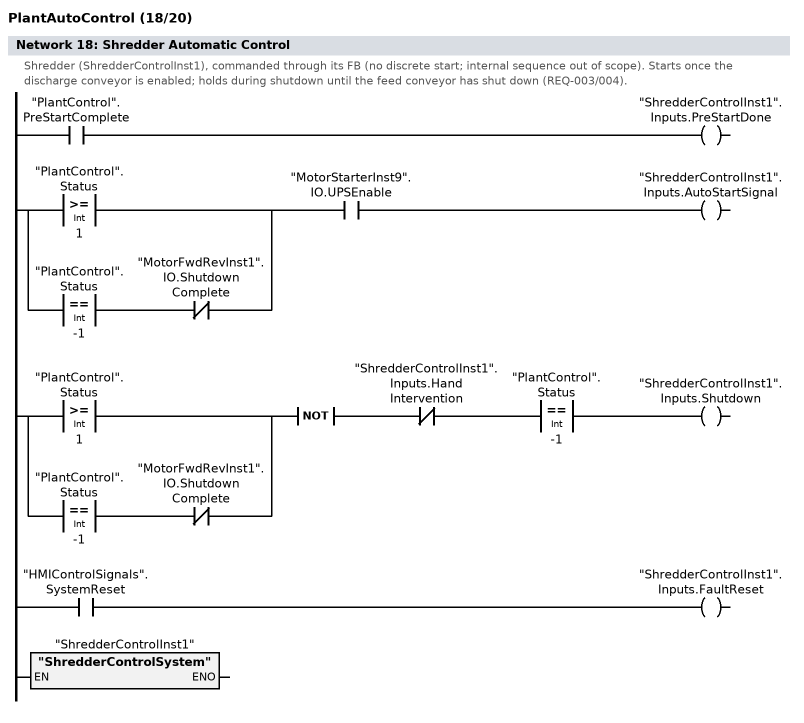
   "ShredderControlInst1".Inputs.PreStartDone := "PlantControl".PreStartComplete;
   "ShredderControlInst1".Inputs.AutoStartSignal := (("PlantControl".Status >= 1) OR (("PlantControl".Status = (-1)) AND NOT "MotorFwdRevInst1".IO.ShutdownComplete)) AND "MotorStarterInst9".IO.UPSEnable;
   "ShredderControlInst1".Inputs.Shutdown := NOT (("PlantControl".Status >= 1) OR (("PlantControl".Status = (-1)) AND NOT "MotorFwdRevInst1".IO.ShutdownComplete)) AND NOT "ShredderControlInst1".Inputs.HandIntervention AND ("PlantControl".Status = (-1));
   "ShredderControlInst1".Inputs.FaultReset := "HMIControlSignals".SystemReset;
   "ShredderControlInst1"();   // "ShredderControlSystem"
END_REGION

REGION Network 19: Cyclone Filter Unit Automatic Control
   // Cyclone filter unit (FilterUnitInst1). Remote-operational feedback and reset brought in; fault taken from the inverse of the system-OK signal (REQ-019). Running feedback NOT wired - its source tag DiscreteInputs.'CycloneDustAutoRunning/Stop' contains a '/' and is un-referenceable in IR (C-005 violation in the given DB); see report. Fan up-to-speed from the plant fan-start time (REQ-020). Runs with the plant; holds until fans-shutdown-ready (REQ-003).
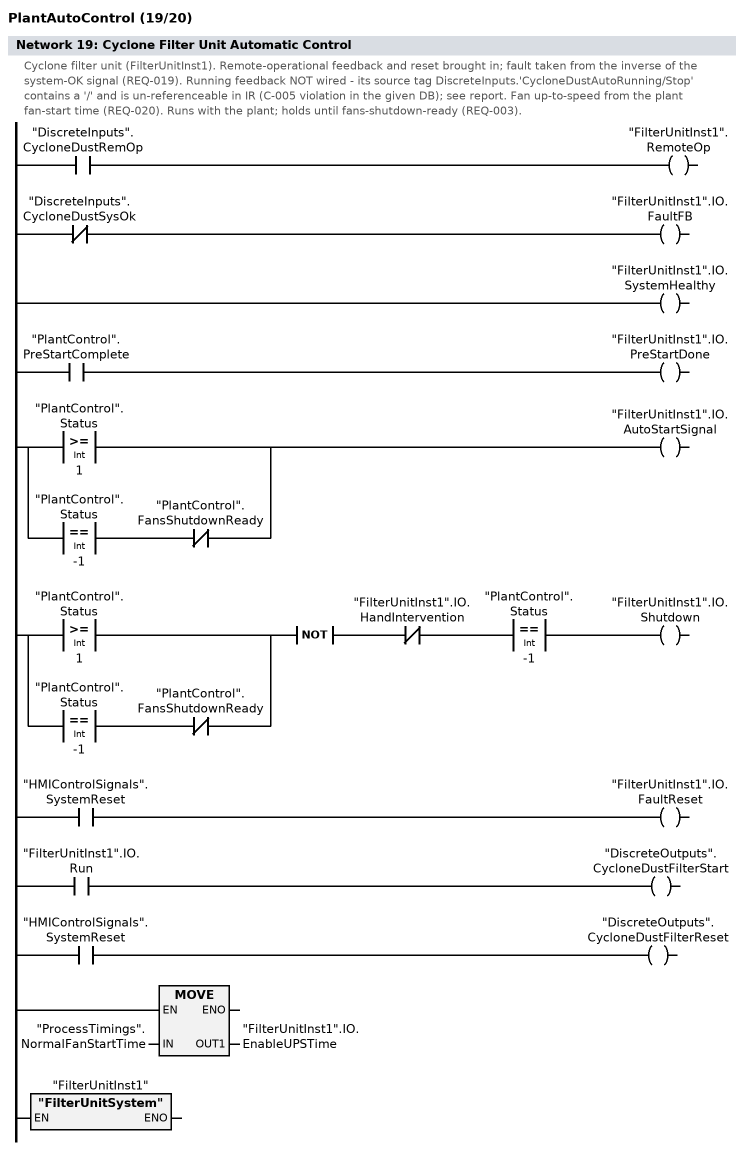
   "FilterUnitInst1".RemoteOp := "DiscreteInputs".CycloneDustRemOp;
   "FilterUnitInst1".IO.FaultFB := NOT "DiscreteInputs".CycloneDustSysOk;
   "FilterUnitInst1".IO.SystemHealthy := TRUE;
   "FilterUnitInst1".IO.PreStartDone := "PlantControl".PreStartComplete;
   "FilterUnitInst1".IO.AutoStartSignal := ("PlantControl".Status >= 1) OR (("PlantControl".Status = (-1)) AND NOT "PlantControl".FansShutdownReady);
   "FilterUnitInst1".IO.Shutdown := NOT (("PlantControl".Status >= 1) OR (("PlantControl".Status = (-1)) AND NOT "PlantControl".FansShutdownReady)) AND NOT "FilterUnitInst1".IO.HandIntervention AND ("PlantControl".Status = (-1));
   "FilterUnitInst1".IO.FaultReset := "HMIControlSignals".SystemReset;
   "DiscreteOutputs".CycloneDustFilterStart := "FilterUnitInst1".IO.Run;
   "DiscreteOutputs".CycloneDustFilterReset := "HMIControlSignals".SystemReset;
   "FilterUnitInst1".IO.EnableUPSTime := "ProcessTimings".NormalFanStartTime;
   "FilterUnitInst1"();   // "FilterUnitSystem"
END_REGION

REGION Network 20: Discharge Conveyor Automatic Control
   // Discharge conveyor (MotorStarterInst9). Gated by the general enable (REQ-013); holds during shutdown until the shredder has shut down (REQ-003).
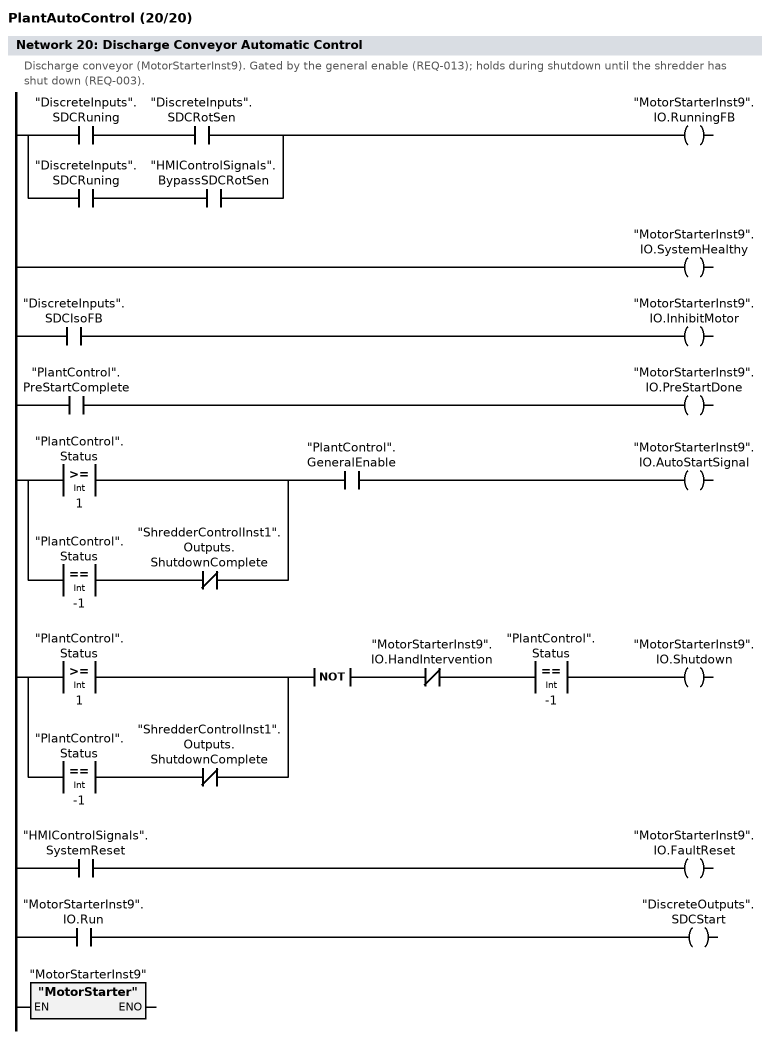
   "MotorStarterInst9".IO.RunningFB := ("DiscreteInputs".SDCRuning AND "DiscreteInputs".SDCRotSen) OR ("DiscreteInputs".SDCRuning AND "HMIControlSignals".BypassSDCRotSen);
   "MotorStarterInst9".IO.SystemHealthy := TRUE;
   "MotorStarterInst9".IO.InhibitMotor := "DiscreteInputs".SDCIsoFB;
   "MotorStarterInst9".IO.PreStartDone := "PlantControl".PreStartComplete;
   "MotorStarterInst9".IO.AutoStartSignal := (("PlantControl".Status >= 1) OR (("PlantControl".Status = (-1)) AND NOT "ShredderControlInst1".Outputs.ShutdownComplete)) AND "PlantControl".GeneralEnable;
   "MotorStarterInst9".IO.Shutdown := NOT (("PlantControl".Status >= 1) OR (("PlantControl".Status = (-1)) AND NOT "ShredderControlInst1".Outputs.ShutdownComplete)) AND NOT "MotorStarterInst9".IO.HandIntervention AND ("PlantControl".Status = (-1));
   "MotorStarterInst9".IO.FaultReset := "HMIControlSignals".SystemReset;
   "DiscreteOutputs".SDCStart := "MotorStarterInst9".IO.Run;
   "MotorStarterInst9"();   // "MotorStarter"
END_REGION
END_FUNCTION
